(* IEC 61131-3 sources: CodesysTest/export/Unused/FB_SimBasicBagDelivery.pou, 3 files *)

(* ---- FB_SimBasicBagDelivery.pou.st ---- *)
(*#-#-#-#-#-#-#-#-#-#---Declaration---#-#-#-#-#-#-#-#-#-#-#-#-#*)

FUNCTION_BLOCK FB_SimBasicBagDelivery EXTENDS FB_BaseComponent IMPLEMENTS IBagDelivery, IExecuteAutomatically
VAR_INPUT
	feedSpeed : UDINT;
	reverseSpeed : UDINT;
	printSpeed : UDINT;
	printLength : REAL;
	bagLength : REAL;
	reverseLength : REAL;
	printOffset : REAL;
END_VAR
VAR_OUTPUT
END_VAR

VAR
	feedAtPrintSpeed : FB_SimulatedFeedback(name := CONCAT(_prefix,'Feed at Print Speed'));
	feedBagOut : FB_SimulatedFeedback(name := CONCAT(_prefix,'Feed Bag Out'));
	feedToPrintOffset : FB_SimulatedFeedback(name := CONCAT(_prefix,'Feed to Print Offset'));
	reverseToSeparate : FB_SimulatedFeedback(name := CONCAT(_prefix,'Reverse to Separate'));
END_VAR
(*#-#-#-#-#-#-#-#-#-#---Implementation---#-#-#-#-#-#-#-#-#-#-#-#-#*)

(* ---- ClearStatus.m.st ---- *)
(*#-#-#-#-#-#-#-#-#-#---Declaration---#-#-#-#-#-#-#-#-#-#-#-#-#*)

METHOD PRIVATE ClearStatus
VAR_INPUT
END_VAR
(*#-#-#-#-#-#-#-#-#-#---Implementation---#-#-#-#-#-#-#-#-#-#-#-#-#*)

feedAtPrintSpeed.in := FALSE;
feedBagOut.in := FALSE;
feedToPrintOffset.in := FALSE;
reverseToSeparate.in := FALSE;
THIS^.Execute();

(* ---- FeedToPhotoeye.m.st ---- *)
(*#-#-#-#-#-#-#-#-#-#---Declaration---#-#-#-#-#-#-#-#-#-#-#-#-#*)

METHOD FeedToPhotoeye
VAR_INPUT
END_VAR
(*#-#-#-#-#-#-#-#-#-#---Implementation---#-#-#-#-#-#-#-#-#-#-#-#-#*)
